// Mitsubishi GX Works2 project: LRI.gx3_ESTADO   PLC: Q03UDV
// V1

PROGRAM MAIN
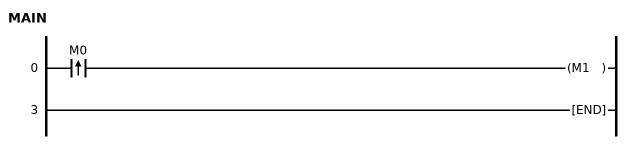
0     LDP     M0
      OUT     M1
3     END
END_PROGRAM
